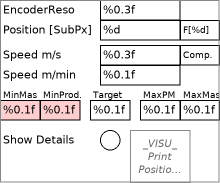
VISUALIZATION _VISU_PmPosition  // 220x183
VAR_IN_OUT
  mInst : FB_PrintModule_WEU;
END_VAR
    RoundedRectangle (0,100 40x20), colour toggle: mInst.bMoving
    RoundedRectangle (40,100 40x20), colour toggle: mInst.bSpeedReachedForPrinting
    RoundedRectangle (140,100 40x20), tooltip "Exeeds max. speed=%f", colour toggle: mInst._pModuleMachineFeedback^.bSpeedExeeded
        p4168582468: mInst._pModuleMachineFeedback^.fMaxSpeed
    RoundedRectangle (180,100 40x20), tooltip "Exeeds max. speed=%f", colour toggle: mInst.fbPrintPosition.fbPositionMaster.fMasterSpeed > mInst.fbPrintPosition.fbPositionMaster.fC_MaxSpeed
    Rectangle (0,0 100x20), "EncoderReso"
    Rectangle (0,45 100x20), "Speed m/s"
    Rectangle (100,45 80x20), "%0.3f", text variable: mInst.fSpeed
    Rectangle (0,65 100x20), "Speed m/min"
    Rectangle (100,65 80x20), "%0.1f", text variable: mInst.fSpeedMpMin, colour toggle: (mInst.fSpeed*60 >= mInst.fC_MinimalProductionSpeed_in_MpMin) AND mInst.fSpeed < mInst._pModuleMachineFeedback^.fMaxSpeed
    Rectangle (0,130 110x20), "Show Details"
    Ellipse (100,130 20x20)
        toggle mInst.fbView.bShowPositionDetail
    Frame (130,130 60x53), invisible if: NOT mInst.fbView.bShowPositionDetail
        shows _VISU_PrintPositionDmax(m_Inst := mInst.fbPrintPosition)
    Rectangle (40,100 40x20), "%0.1f", tooltip "Min. Speed for Production", text variable: mInst.fC_MinimalProductionSpeed_in_MpMin
    Rectangle (100,0 80x20), "%0.3f", text variable: mInst.fbPrintPosition._fEncoderResolution
    Rectangle (0,20 100x20), "Position [SubPx]"
    Rectangle (100,20 80x20), "%d", text variable: mInst.nPos_SubPx
    RoundedRectangle (180,20 40x20), "F[%d]", tooltip "encoder filter active", text variable: mInst.fbPrintPosition.fbPositionMaster.nFilterDepth, colour toggle: mInst.fbPrintPosition.fbPositionMaster.bEnableFilter, invisible if: NOT mInst.fbPrintPosition.fbPositionMaster.bEnableFilter
    RoundedRectangle (180,45 40x20), "Comp.", tooltip "encoder filter active", colour toggle: mInst.fbPrintPosition._bEnSpeedComp, invisible if: NOT mInst.fbPrintPosition._bEnSpeedComp
    Rectangle (0,100 40x20), "%0.1f", tooltip "Min. Speed for Production", text variable: mInst.fbPrintPosition.fbPositionMaster.fC_MinSpeed*60
    Rectangle (180,100 40x20), "%0.1f", tooltip "Min. Speed for Production", text variable: mInst.fbPrintPosition.fbPositionMaster.fC_MaxSpeed*60
    Rectangle (140,100 40x20), "%0.1f", tooltip "Min. Speed for Production", text variable: mInst._pModuleMachineFeedback^.fMaxSpeed
    Rectangle (0,85 40x20), "MinMas"
    Rectangle (40,85 40x20), "MinProd."
    Rectangle (140,85 40x20), "MaxPM"
    Rectangle (180,85 40x20), "MaxMas"
    Rectangle (90,85 40x20), "Target"
    Rectangle (90,100 40x20), "%0.1f", tooltip "Min. Speed for Production", text variable: mInst._pModuleMachineState^.fTargetSpeed*60
END_VISUALIZATION

(* stored: Version 1.1.0.1, ProductVersion 3.1.4024.11
   Visu _VISU_PmPosition: Id {b3e81474-f053-4071-9e52-4e6308952c25} *)
